// TIA Portal V20 export
FUNCTION_BLOCK "FB - Sabload"   // FB5, LAD
TITLE = Equipment - Sabload
{ S7_Optimized_Access := 'TRUE' }
// This function block contains all logic for controlling a Sabload module.
// -This module consists of a jig, table, airbag part detection layser sensors.
// 
// >> Block created by: Engr. Awais Ali
// >> Block creation date:  08-10-2025
// stored: MemoryReserve 100, SetENOAutomatically false
   VAR_INPUT
      i_xPart1 : Bool;
      i_xPart2 : Bool;
      i_xPart3 : Bool;
      i_xPart4 : Bool;
   END_VAR
   VAR_IN_OUT
      iq_Sabload : "UDT-SABload";
      iq_Tablecheck : "UDT-TableCheck";
   END_VAR
   VAR
      iState : Int;
      OndelayJigPresent { S7_SetPoint := 'True'} : TON_TIME;
      OnDelayPart1 { S7_SetPoint := 'True'} : TON_TIME;
      OnDelayPart2 { S7_SetPoint := 'True'} : TON_TIME;
      OnDelayPart3 { S7_SetPoint := 'True'} : TON_TIME;
      OnDelayPart4 { S7_SetPoint := 'True'} : TON_TIME;
      TriggerS1 : Bool;
      OnDelayReset { S7_SetPoint := 'True'} : TON_TIME;
      TriggerS6 : Bool;
      TriggerS2 { ExternalAccessible := 'False'; ExternalVisible := 'False'; ExternalWritable := 'False'} : Bool;
      TriggerS3 { ExternalAccessible := 'False'; ExternalVisible := 'False'; ExternalWritable := 'False'} : Bool;
      TriggerS4 { ExternalAccessible := 'False'; ExternalVisible := 'False'; ExternalWritable := 'False'} : Bool;
      TriggerS5 { ExternalAccessible := 'False'; ExternalVisible := 'False'; ExternalWritable := 'False'} : Bool;
      Oneshot_IndicationLamp { S7_SetPoint := 'True'} : TP_TIME;
      OnDelay_fault1 { S7_SetPoint := 'True'} : TON_TIME;
      OnDelayPart5 { S7_SetPoint := 'True'} : TON_TIME;
      InstanceTrigger_part1 { S7_SetPoint := 'True'} : R_TRIG;
      InstanceTrigger_part2 { S7_SetPoint := 'True'} : R_TRIG;
      InstanceTrigger_part3 { S7_SetPoint := 'True'} : R_TRIG;
      InstanceTrigger_part4 { S7_SetPoint := 'True'} : R_TRIG;
      xOkPart : Bool;
      xpartOrderComplete : Bool;
      Instance_F_trigger_part1 { S7_SetPoint := 'True'} : F_TRIG;
   END_VAR
   VAR_TEMP   // added for the SCL form of the ladder/FBD networks
      _w1 : Bool;
   END_VAR
BEGIN

REGION Network 1: Control - part one
   // if the 1st part place on the Jig for x seconds the state move from 0 to 5. It confirm the part is there.
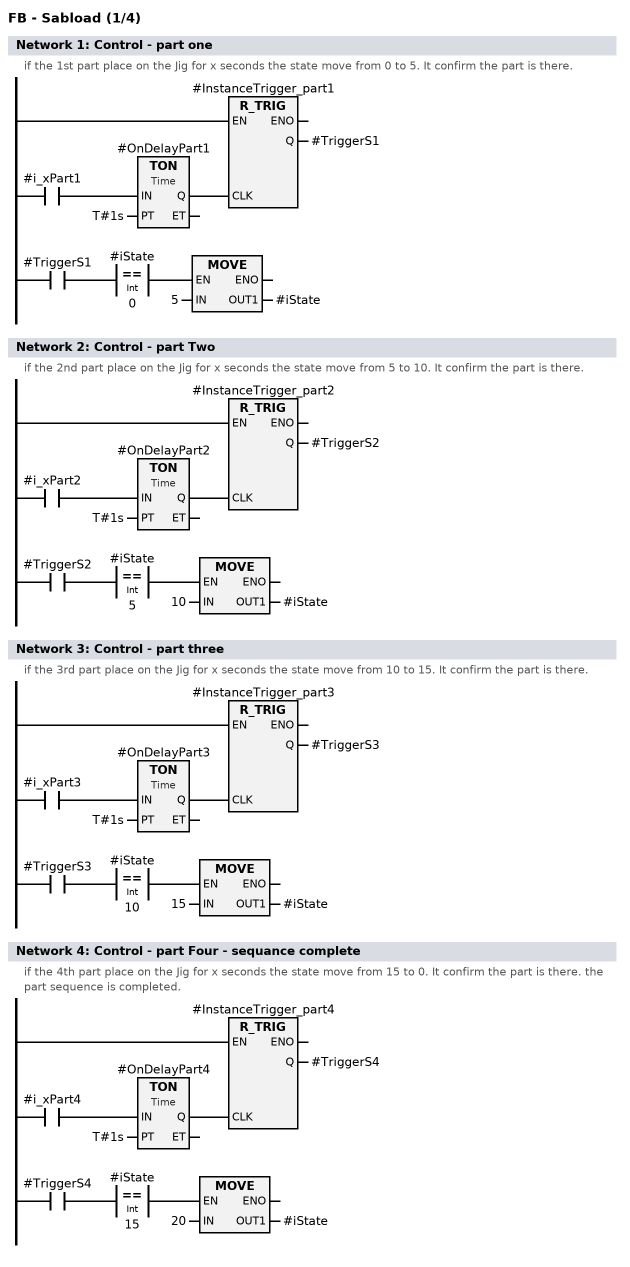
   RUNG wire#powerrail
      #InstanceTrigger_part1.R_TRIG(CLK := wire#w1, Q => #TriggerS1)
   END_RUNG
   RUNG wire#powerrail
      Contact( #i_xPart1 )
      { S7_Templates := "time_type := Time" } #OnDelayPart1.TON(pt := T#1s, et =>)
   END_RUNG wire#w1
   RUNG wire#powerrail
      Contact( #TriggerS1 )
      { S7_Templates := "SrcType := Int" } EQ_Contact(in1 := #iState, in2 := 0)
      Move(in := 5, out1 => #iState)
   END_RUNG
   // the same network as SCL:
   #OnDelayPart1(IN := #i_xPart1, PT := T#1s);   // TON
   #InstanceTrigger_part1(CLK := #OnDelayPart1.Q, Q => #TriggerS1);   // R_TRIG
   IF #TriggerS1 AND (#iState = 0) THEN #iState := 5; END_IF;
END_REGION

REGION Network 2: Control - part Two
   // if the 2nd part place on the Jig for x seconds the state move from 5 to 10. It confirm the part is there.
   RUNG wire#powerrail
      #InstanceTrigger_part2.R_TRIG(CLK := wire#w1, Q => #TriggerS2)
   END_RUNG
   RUNG wire#powerrail
      Contact( #i_xPart2 )
      { S7_Templates := "time_type := Time" } #OnDelayPart2.TON(pt := T#1s, et =>)
   END_RUNG wire#w1
   RUNG wire#powerrail
      Contact( #TriggerS2 )
      { S7_Templates := "SrcType := Int" } EQ_Contact(in1 := #iState, in2 := 5)
      Move(in := 10, out1 => #iState)
   END_RUNG
   // the same network as SCL:
   #OnDelayPart2(IN := #i_xPart2, PT := T#1s);   // TON
   #InstanceTrigger_part2(CLK := #OnDelayPart2.Q, Q => #TriggerS2);   // R_TRIG
   IF #TriggerS2 AND (#iState = 5) THEN #iState := 10; END_IF;
END_REGION

REGION Network 3: Control - part three
   // if the 3rd part place on the Jig for x seconds the state move from 10 to 15. It confirm the part is there.
   RUNG wire#powerrail
      #InstanceTrigger_part3.R_TRIG(CLK := wire#w1, Q => #TriggerS3)
   END_RUNG
   RUNG wire#powerrail
      Contact( #i_xPart3 )
      { S7_Templates := "time_type := Time" } #OnDelayPart3.TON(pt := T#1s, et =>)
   END_RUNG wire#w1
   RUNG wire#powerrail
      Contact( #TriggerS3 )
      { S7_Templates := "SrcType := Int" } EQ_Contact(in1 := #iState, in2 := 10)
      Move(in := 15, out1 => #iState)
   END_RUNG
   // the same network as SCL:
   #OnDelayPart3(IN := #i_xPart3, PT := T#1s);   // TON
   #InstanceTrigger_part3(CLK := #OnDelayPart3.Q, Q => #TriggerS3);   // R_TRIG
   IF #TriggerS3 AND (#iState = 10) THEN #iState := 15; END_IF;
END_REGION

REGION Network 4: Control - part Four - sequance complete
   // if the 4th part place on the Jig for x seconds the state move from 15 to 0. It confirm the part is there. the part sequence is completed.
   RUNG wire#powerrail
      #InstanceTrigger_part4.R_TRIG(CLK := wire#w1, Q => #TriggerS4)
   END_RUNG
   RUNG wire#powerrail
      Contact( #i_xPart4 )
      { S7_Templates := "time_type := Time" } #OnDelayPart4.TON(pt := T#1s, et =>)
   END_RUNG wire#w1
   RUNG wire#powerrail
      Contact( #TriggerS4 )
      { S7_Templates := "SrcType := Int" } EQ_Contact(in1 := #iState, in2 := 15)
      Move(in := 20, out1 => #iState)
   END_RUNG
   // the same network as SCL:
   #OnDelayPart4(IN := #i_xPart4, PT := T#1s);   // TON
   #InstanceTrigger_part4(CLK := #OnDelayPart4.Q, Q => #TriggerS4);   // R_TRIG
   IF #TriggerS4 AND (#iState = 15) THEN #iState := 20; END_IF;
END_REGION

REGION Network 5: Control - Remove the jig: sequance complete
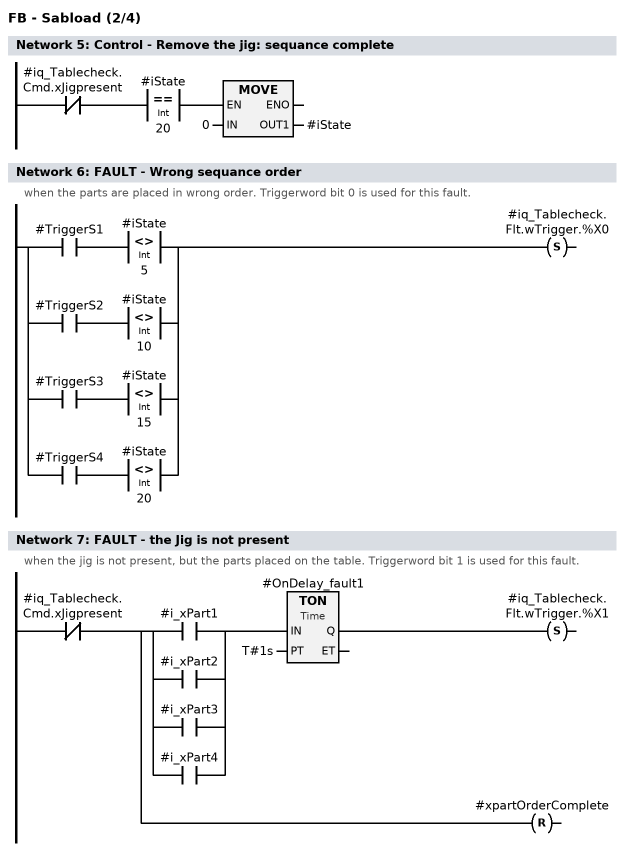
   RUNG wire#powerrail
      I_Contact( #iq_Tablecheck.Cmd.xJigpresent )
      { S7_Templates := "SrcType := Int" } EQ_Contact(in1 := #iState, in2 := 20)
      Move(in := 0, out1 => #iState)
   END_RUNG
   // the same network as SCL:
   IF NOT #iq_Tablecheck.Cmd.xJigpresent AND (#iState = 20) THEN #iState := 0; END_IF;
END_REGION

REGION Network 6: FAULT - Wrong sequance order
   // when the parts are placed in wrong order. Triggerword bit 0 is used for this fault.
   RUNG wire#powerrail
      Contact( #TriggerS1 )
      { S7_Templates := "SrcType := Int" } NE_Contact(in1 := #iState, in2 := 5)
      wire#w1
      S_Coil( #iq_Tablecheck.Flt.wTrigger.%X0 )
   END_RUNG
   RUNG wire#powerrail
      Contact( #TriggerS2 )
      { S7_Templates := "SrcType := Int" } NE_Contact(in1 := #iState, in2 := 10)
   END_RUNG wire#w1
   RUNG wire#powerrail
      Contact( #TriggerS3 )
      { S7_Templates := "SrcType := Int" } NE_Contact(in1 := #iState, in2 := 15)
   END_RUNG wire#w1
   RUNG wire#powerrail
      Contact( #TriggerS4 )
      { S7_Templates := "SrcType := Int" } NE_Contact(in1 := #iState, in2 := 20)
   END_RUNG wire#w1
   // the same network as SCL:
   IF (#TriggerS1 AND (#iState <> 5)) OR (#TriggerS2 AND (#iState <> 10)) OR (#TriggerS3 AND (#iState <> 15)) OR (#TriggerS4 AND (#iState <> 20)) THEN
       #iq_Tablecheck.Flt.wTrigger.%X0 := TRUE;
   END_IF;
END_REGION

REGION Network 7: FAULT - the Jig is not present
   // when the jig is not present, but the parts placed on the table. Triggerword bit 1 is used for this fault.
   RUNG wire#powerrail
      I_Contact( #iq_Tablecheck.Cmd.xJigpresent )
      wire#w1
      Contact( #i_xPart1 )
      wire#w2
      { S7_Templates := "time_type := Time" } #OnDelay_fault1.TON(pt := T#1s, et =>)
      S_Coil( #iq_Tablecheck.Flt.wTrigger.%X1 )
   END_RUNG
   RUNG wire#w1
      Contact( #i_xPart2 )
   END_RUNG wire#w2
   RUNG wire#w1
      Contact( #i_xPart3 )
   END_RUNG wire#w2
   RUNG wire#w1
      Contact( #i_xPart4 )
   END_RUNG wire#w2
   RUNG wire#w1
      R_Coil( #xpartOrderComplete )
   END_RUNG
   // the same network as SCL:
   #_w1 := NOT #iq_Tablecheck.Cmd.xJigpresent;
   #OnDelay_fault1(IN := #_w1 AND (#i_xPart1 OR #i_xPart2 OR #i_xPart3 OR #i_xPart4), PT := T#1s);   // TON
   IF #OnDelay_fault1.Q THEN #iq_Tablecheck.Flt.wTrigger.%X1 := TRUE; END_IF;
   IF #_w1 THEN #xpartOrderComplete := FALSE; END_IF;
END_REGION

REGION Network 8: FAULT - previous parts missing
   // when the palced parts removed before completing the sequnace. Triggerword bit 1 is used for this fault.
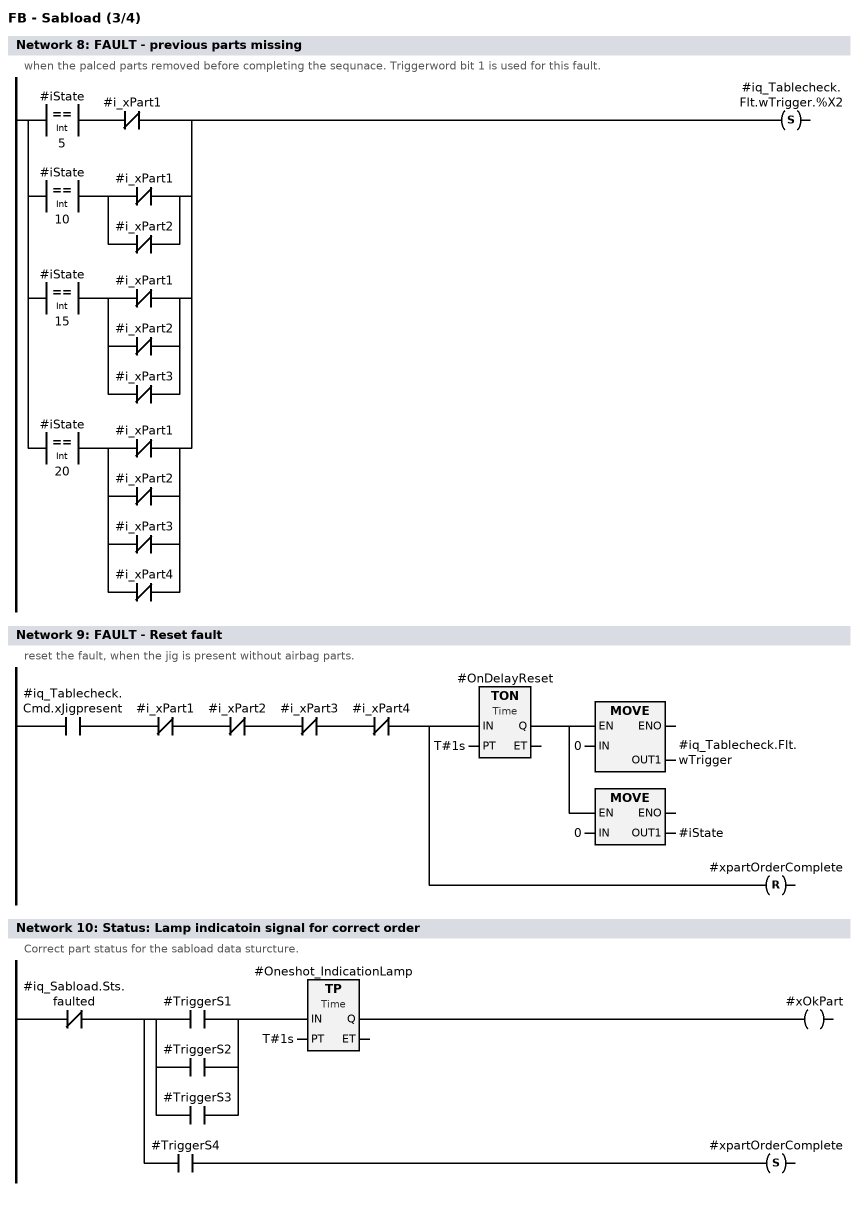
   RUNG wire#powerrail
      { S7_Templates := "SrcType := Int" } EQ_Contact(in1 := #iState, in2 := 5)
      I_Contact( #i_xPart1 )
      wire#w1
      S_Coil( #iq_Tablecheck.Flt.wTrigger.%X2 )
   END_RUNG
   RUNG wire#powerrail
      { S7_Templates := "SrcType := Int" } EQ_Contact(in1 := #iState, in2 := 10)
      wire#w2
      I_Contact( #i_xPart1 )
   END_RUNG wire#w1
   RUNG wire#w2
      I_Contact( #i_xPart2 )
   END_RUNG wire#w1
   RUNG wire#powerrail
      { S7_Templates := "SrcType := Int" } EQ_Contact(in1 := #iState, in2 := 15)
      wire#w3
      I_Contact( #i_xPart1 )
   END_RUNG wire#w1
   RUNG wire#w3
      I_Contact( #i_xPart2 )
   END_RUNG wire#w1
   RUNG wire#w3
      I_Contact( #i_xPart3 )
   END_RUNG wire#w1
   RUNG wire#powerrail
      { S7_Templates := "SrcType := Int" } EQ_Contact(in1 := #iState, in2 := 20)
      wire#w4
      I_Contact( #i_xPart1 )
   END_RUNG wire#w1
   RUNG wire#w4
      I_Contact( #i_xPart2 )
   END_RUNG wire#w1
   RUNG wire#w4
      I_Contact( #i_xPart3 )
   END_RUNG wire#w1
   RUNG wire#w4
      I_Contact( #i_xPart4 )
   END_RUNG wire#w1
   // the same network as SCL:
   IF ((#iState = 5) AND NOT #i_xPart1) OR ((#iState = 10) AND (NOT #i_xPart1 OR NOT #i_xPart2)) OR ((#iState = 15) AND (NOT #i_xPart1 OR NOT #i_xPart2 OR NOT #i_xPart3)) OR ((#iState = 20) AND (NOT #i_xPart1 OR NOT #i_xPart2 OR NOT #i_xPart3 OR NOT #i_xPart4)) THEN
       #iq_Tablecheck.Flt.wTrigger.%X2 := TRUE;
   END_IF;
END_REGION

REGION Network 9: FAULT - Reset fault
   // reset the fault, when the jig is present without airbag parts.
   RUNG wire#powerrail
      Contact( #iq_Tablecheck.Cmd.xJigpresent )
      I_Contact( #i_xPart1 )
      I_Contact( #i_xPart2 )
      I_Contact( #i_xPart3 )
      I_Contact( #i_xPart4 )
      wire#w1
      { S7_Templates := "time_type := Time" } #OnDelayReset.TON(pt := T#1s, et =>)
      wire#w2
      Move(in := 0, out1 => #iq_Tablecheck.Flt.wTrigger)
   END_RUNG
   RUNG wire#w2
      Move(in := 0, out1 => #iState)
   END_RUNG
   RUNG wire#w1
      R_Coil( #xpartOrderComplete )
   END_RUNG
   // the same network as SCL:
   #_w1 := #iq_Tablecheck.Cmd.xJigpresent AND NOT #i_xPart1 AND NOT #i_xPart2 AND NOT #i_xPart3 AND NOT #i_xPart4;
   #OnDelayReset(IN := #_w1, PT := T#1s);   // TON
   IF #OnDelayReset.Q THEN
       #iq_Tablecheck.Flt.wTrigger := 0;
       #iState := 0;
   END_IF;
   IF #_w1 THEN #xpartOrderComplete := FALSE; END_IF;
END_REGION

REGION Network 10: Status: Lamp indicatoin signal for correct order
   // Correct part status for the sabload data sturcture.
   RUNG wire#powerrail
      I_Contact( #iq_Sabload.Sts.faulted )
      wire#w1
      Contact( #TriggerS1 )
      wire#w2
      { S7_Templates := "time_type := Time" } #Oneshot_IndicationLamp.TP(pt := T#1s, et =>)
      Coil( #xOkPart )
   END_RUNG
   RUNG wire#w1
      Contact( #TriggerS2 )
   END_RUNG wire#w2
   RUNG wire#w1
      Contact( #TriggerS3 )
   END_RUNG wire#w2
   RUNG wire#w1
      Contact( #TriggerS4 )
      S_Coil( #xpartOrderComplete )
   END_RUNG
   // the same network as SCL:
   #_w1 := NOT #iq_Sabload.Sts.faulted;
   #Oneshot_IndicationLamp(IN := #_w1 AND (#TriggerS1 OR #TriggerS2 OR #TriggerS3), PT := T#1s);   // TP
   #xOkPart := #Oneshot_IndicationLamp.Q;
   IF #_w1 AND #TriggerS4 THEN #xpartOrderComplete := TRUE; END_IF;
END_REGION

REGION Network 11: the part of the airbage is placed correctly
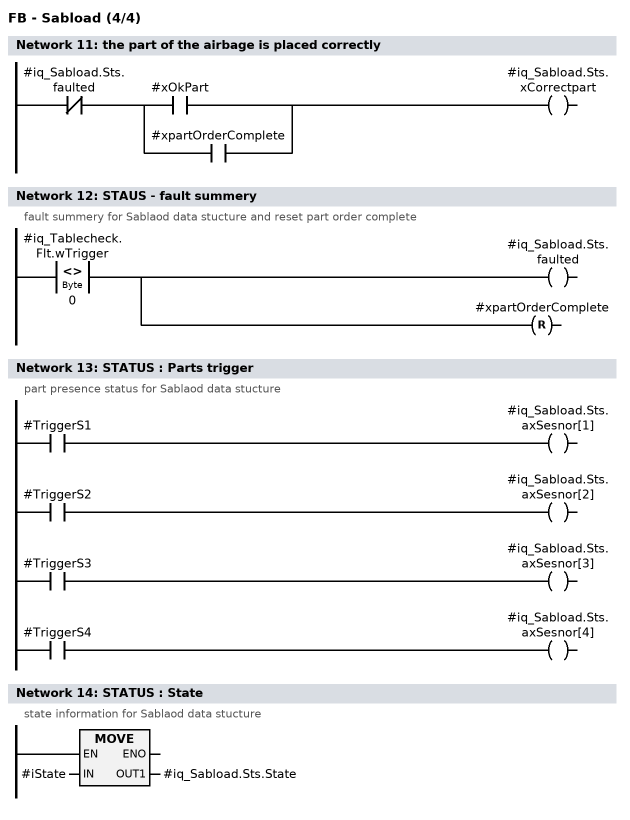
   RUNG wire#powerrail
      I_Contact( #iq_Sabload.Sts.faulted )
      wire#w1
      Contact( #xOkPart )
      wire#w2
      Coil( #iq_Sabload.Sts.xCorrectpart )
   END_RUNG
   RUNG wire#w1
      Contact( #xpartOrderComplete )
   END_RUNG wire#w2
   // the same network as SCL:
   #iq_Sabload.Sts.xCorrectpart := NOT #iq_Sabload.Sts.faulted AND (#xOkPart OR #xpartOrderComplete);
END_REGION

REGION Network 12: STAUS - fault summery
   // fault summery for Sablaod data stucture and reset part order complete
   RUNG wire#powerrail
      { S7_Templates := "SrcType := Byte" } NE_Contact(in1 := #iq_Tablecheck.Flt.wTrigger, in2 := 0)
      wire#w1
      Coil( #iq_Sabload.Sts.faulted )
   END_RUNG
   RUNG wire#w1
      R_Coil( #xpartOrderComplete )
   END_RUNG
   // the same network as SCL:
   #iq_Sabload.Sts.faulted := #iq_Tablecheck.Flt.wTrigger <> 0;
   IF #iq_Sabload.Sts.faulted THEN #xpartOrderComplete := FALSE; END_IF;
END_REGION

REGION Network 13: STATUS : Parts trigger
   // part presence status for Sablaod data stucture
   RUNG wire#powerrail
      Contact( #TriggerS1 )
      Coil( #iq_Sabload.Sts.axSesnor[1] )
   END_RUNG
   RUNG wire#powerrail
      Contact( #TriggerS2 )
      Coil( #iq_Sabload.Sts.axSesnor[2] )
   END_RUNG
   RUNG wire#powerrail
      Contact( #TriggerS3 )
      Coil( #iq_Sabload.Sts.axSesnor[3] )
   END_RUNG
   RUNG wire#powerrail
      Contact( #TriggerS4 )
      Coil( #iq_Sabload.Sts.axSesnor[4] )
   END_RUNG
   // the same network as SCL:
   #iq_Sabload.Sts.axSesnor[1] := #TriggerS1;
   #iq_Sabload.Sts.axSesnor[2] := #TriggerS2;
   #iq_Sabload.Sts.axSesnor[3] := #TriggerS3;
   #iq_Sabload.Sts.axSesnor[4] := #TriggerS4;
END_REGION

REGION Network 14: STATUS : State
   // state information for Sablaod data stucture
   RUNG wire#powerrail
      Move(in := #iState, out1 => #iq_Sabload.Sts.State)
   END_RUNG
   // the same network as SCL:
   #iq_Sabload.Sts.State := #iState;
END_REGION
END_FUNCTION_BLOCK
